PROGRAM P_Divisao
VAR
	bCalcular	: BOOL;
	rValor1		: REAL;
	rValor2		: REAL;
	rResultado	: REAL;
END_VAR

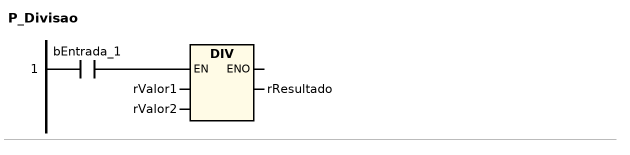
// NETWORK 1
IF bEntrada_1 THEN rResultado := rValor1 / rValor2; END_IF

END_PROGRAM

(* stored: Version 1.1.0.1, ProductVersion 3.1.4024.12
   POU P_Divisao: Id {646dad23-e2ee-4c54-9081-42b14f52b44d}, SpecialFunc None *)
